INTERFACE I_CoE_property

PROPERTY CoE_communication_handler : I_CoE_communication_handler
GET
END_GET
SET
END_SET
END_PROPERTY

PROPERTY dataTypeSize : UDINT
GET
END_GET
END_PROPERTY

METHOD get_value : BOOL
VAR_OUTPUT
    value : Tc2_Utilities.T_Arg ;
	errId : UDINT;
END_VAR
END_METHOD

METHOD handle_read_callback : BOOL
VAR_INPUT
	pt_buffer : POINTER TO Tc2_Utilities.T_Arg;
	errId : UDINT;
END_VAR
END_METHOD

METHOD handle_write_callback : BOOL
VAR_INPUT
	errId : UDINT;
END_VAR
END_METHOD

PROPERTY Index : word
GET
END_GET
END_PROPERTY

PROPERTY init_done : bool
GET
END_GET
END_PROPERTY

PROPERTY PropertyType : E_ArgType
GET
END_GET
SET
END_SET
END_PROPERTY

(**
This method is initializing or reinitializing the property and returns TRUE when this is done.
In case of an error during the init it returns the ErrorCode related to the error that occurred.
*)
METHOD reinit : BOOL
VAR_OUTPUT
	errId: UDINT;
END_VAR
END_METHOD

METHOD run : BOOL
VAR_INPUT
END_VAR
END_METHOD

METHOD set_value : BOOL
VAR_INPUT
    value : Tc2_Utilities.T_Arg ;
END_VAR
END_METHOD

PROPERTY SlaveAddress : UINT
GET
END_GET
SET
END_SET
END_PROPERTY

PROPERTY SubIndex : BYTE
GET
END_GET
END_PROPERTY

PROPERTY valueToWrite : Tc2_Utilities.T_Arg
GET
END_GET
END_PROPERTY

END_INTERFACE

(* stored: Version 1.1.0.1, ProductVersion 3.1.4024.9
   Itf I_CoE_property: Id {7c1857e7-bee5-07f1-0b20-6cf74deec630}
   Property CoE_communication_handler: Id {91922664-d8dd-07af-3101-9d6e03189e03}
   Get Get: Id {33e63e6b-9402-0002-3803-52403f88ffa7}
   Set Set: Id {50ad2432-1f12-06bc-0caa-410833dc60a8}
   Property dataTypeSize: Id {de387db6-9200-03b5-04ce-c696adad2786}
   Get Get: Id {d1bf6bb7-1fae-0c67-2a89-9b9671a3ed40}
   Method get_value: Id {a61ec230-9e45-0e05-0075-8d4d5f019271}
   Method handle_read_callback: Id {f97bb7a1-54c0-0520-2966-3954b2ce9d96}
   Method handle_write_callback: Id {4711a839-42f9-0006-20a7-8f6c7c920378}
   Property Index: Id {9508ced1-8e4a-0a57-111a-73fd015de83e}
   Get Get: Id {c674f8d0-a3dd-01cf-25ff-3766a9746bed}
   Property init_done: Id {899acaec-934e-0006-179c-e29da311289d}
   Get Get: Id {8fb5aeb2-7d17-0a65-17c2-6df7951761f2}
   Property PropertyType: Id {5b4ff985-3b5b-043d-0f69-1d2015775354}
   Get Get: Id {3b990a39-4f53-0970-37d3-f413b06d4805}
   Set Set: Id {c3c90df5-9d83-0e15-37d7-c1d8916c5ec5}
   Method reinit: Id {e0cf676b-bdca-01f3-3233-1894d274fc8f}
   Method run: Id {f131b58c-bde9-09c5-32c1-30fd69bb6db7}
   Method set_value: Id {494becd6-378b-0798-2ac9-1d7d375f7b0f}
   Property SlaveAddress: Id {89c1fe58-92a8-0d41-0ac4-d20f5c5cbc33}
   Get Get: Id {0e74ced1-ef9d-0777-16a1-2ca34a2c6040}
   Set Set: Id {bd601182-a073-0f2e-146e-a99d19e9bd54}
   Property SubIndex: Id {f509e4a6-fa46-0f01-30c0-69456455fcf5}
   Get Get: Id {63318d45-76d3-0cb2-38d8-67ff2123b9b2}
   Property valueToWrite: Id {3db24a19-dda7-0bad-0dfa-160770f43209}
   Get Get: Id {1b5edc05-7c6e-0691-3b7b-2ed784d430c5} *)
